PROGRAM MAIN
VAR
	fb_rfid : FB_BF_IDM25_SIMPLE;
	fb_id_list : FB_ID_list_man;
	
	local_user_id	: stUserID;
	local_user_list	: ARRAY [0..19] OF stUserID;
END_VAR


// update HMI var here ...
_14_STATE();

fb_rfid(rfid_hw:=GVL.rfid);
fb_id_list(	stUserIn := ADR(local_user_id),
			stArrList := ADR(local_user_list),
			xAdd := HMI.xAddUser.rtrig,
			xDel := HMI.xDelUser.rtrig,
			xAccess := HMI.xFALSE,
			tRestore := T#5S,
			tTimeOut := T#20M);

END_PROGRAM

(* stored: Version 1.1.0.1, ProductVersion 3.1.4024.6
   POU MAIN: Id {3e2d624b-4f29-4b41-b9b7-092210ac80e5}, SpecialFunc None *)
